(* IEC 61131-3 sources: testLang/lang, 1 file *)

(* ---- 1.st ---- *)
PROGRAM ExampleProgram
VAR
    input1 AT %IX0.0 : BOOL;
    output1 AT %QX0.0 : BOOL;
END_VAR

IF input1 THEN
    output1 := TRUE;
ELSE
    output1 := FALSE;
END_IF

	'keyword': [
		/\b(?:END_)?(?:PROGRAM|CONFIGURATION|INTERFACE|FUNCTION_BLOCK|FUNCTION|ACTION|TRANSITION|TYPE|STRUCT|(?:INITIAL_)?STEP|NAMESPACE|LIBRARY|CHANNEL|FOLDER|RESOURCE|VAR_(?:ACCESS|CONFIG|EXTERNAL|GLOBAL|INPUT|IN_OUT|OUTPUT|TEMP)|VAR|METHOD|PROPERTY)\b/i,
		/\b(?:AT|BY|(?:END_)?(?:CASE|FOR|IF|REPEAT|WHILE)|CONSTANT|CONTINUE|DO|ELSE|ELSIF|EXIT|EXTENDS|FROM|GET|GOTO|IMPLEMENTS|JMP|NON_RETAIN|OF|PRIVATE|PROTECTED|PUBLIC|RETAIN|RETURN|SET|TASK|THEN|TO|UNTIL|USING|WITH|__CATCH|__ENDTRY|__FINALLY|__TRY)\b/
	],
	'class-name': /\b(?:ANY|ARRAY|BOOL|BYTE|U?(?:D|L|S)?INT|(?:D|L)?WORD|DATE(?:_AND_TIME)?|DT|L?REAL|POINTER|STRING|TIME(?:_OF_DAY)?|TOD)\b/,
	'address': {
		pattern: /%[IQM][XBWDL][\d.]*|%[IQ][\d.]*/,
		alias: 'symbol'
	},
	'number': /\b(?:16#[\da-f]+|2#[01_]+|0x[\da-f]+)\b|\b(?:D|DT|T|TOD)#[\d_shmd:]*|\b[A-Z]*#[\d.,_]*|(?:\b\d+(?:\.\d*)?|\B\.\d+)(?:e[+-]?\d+)?/i,
	'boolean': /\b(?:FALSE|NULL|TRUE)\b/,
	'operator': /S?R?:?=>?|&&?|\*\*?|<[=>]?|>=?|[-:^/+#]|\b(?:AND|EQ|EXPT|GE|GT|LE|LT|MOD|NE|NOT|OR|XOR)\b/,
	'function': /\b[a-z_]\w*(?=\s*\()/i,
	'punctuation': /[()[\].,;]/,
};
